FUNCTION_BLOCK ConveyorLL
VAR
	enable AT %Q* : BOOL := TRUE;
	direction AT %Q* : BOOL; //FALSE = forward, TRUE = backward
	pulse AT %Q* : BOOL;
	reset AT %Q* : BOOL;
	
	sensorEntry AT %I* : BOOL;
	sensorExit AT %I* : BOOL;

	lifterEnable AT %Q* : BOOL := TRUE;
	lifterDirection AT %Q* : BOOL; //FALSE = up, TRUE = down
	lifterPulse AT %Q* : BOOL;
	lifterReset AT %Q* : BOOL;
END_VAR
VAR_OUTPUT
	operation : ConveyorMode;
	request : ConveyorMode;
	
	error AT %I* : BOOL;
	lifterError AT %I* : BOOL;
	
	position AT %I* : REAL;
	velocity AT %I* : REAL;
	
	hasLifter : BOOL;
	extended AT %I* : BOOL;
	retracted AT %I* : BOOL;
END_VAR
VAR
	nextConveyor : POINTER TO Conveyor;
	prevConveyor : POINTER TO Conveyor;
	
	lifterMode : (HOLD, LIFTER_EXTEND, LIFTER_RETRACT); 
	
	//pulses are assumed to be low-high-low
	pulser : TP;
	lifterPulser : TP;
END_VAR
VAR_STAT CONSTANT
	pulseWidth : TIME := T#25MS;
END_VAR

pulser(IN:= , PT:= pulseWidth, Q=> pulse, ET=> );
pulser.IN := 
	enable AND 
	NOT error AND 
	NOT reset AND 
	(operation = ConveyorMode.FORWARD OR operation = ConveyorMode.BACKWARD)
	AND pulser.Q; //ends pulse itself

lifterPulser(IN:= , PT:= pulseWidth, Q=> lifterPulse, ET=> );
lifterPulser.IN := 
	hasLifter AND
	lifterEnable AND 
	NOT lifterError AND 
	NOT lifterReset AND 
	( (lifterMode = LIFTER_EXTEND AND NOT extended) OR (lifterMode = LIFTER_RETRACT AND NOT retracted) ) AND
	lifterPulser.Q; //self-ending pulse

override();

CASE lifterMode OF
	HOLD:
		lifterDirection := TRUE;
		lifterPulse := FALSE;
		
	LIFTER_EXTEND:
		lifterDirection := FALSE;
		lifterPulse := NOT lifterPulse;
	
	LIFTER_RETRACT:
		lifterDirection := TRUE;
		lifterPulse := NOT lifterPulse;
	
END_CASE

sequence();

METHOD backward : BOOL
VAR_INPUT
END_VAR
END_METHOD

METHOD extend : BOOL
VAR_INPUT
END_VAR
VAR
	noLifter : BOOL;
END_VAR
IF hasLifter THEN
	lifterMode := UP;
	extend := TRUE;
ELSE
	noLifter := TRUE;
END_IF
END_METHOD

METHOD forward : BOOL
VAR_INPUT
END_VAR
END_METHOD

PROPERTY IsOccupied : BOOL
GET
IsOccupied := sensorExit OR sensorEntry;
END_GET
END_PROPERTY

METHOD PRIVATE override : BOOL
VAR_INPUT
END_VAR
IF
	(extended AND lifterMode = UP) OR
	(retracted AND lifterMode = DOWN)
THEN
	lifterMode := HOLD;
END_IF
END_METHOD

METHOD reset : BOOL
VAR_INPUT
END_VAR
position := 0;
velocity := velocity; //no change

extend();
END_METHOD

METHOD retract : BOOL
VAR_INPUT
END_VAR
VAR
	noLifter : BOOL;
END_VAR
IF hasLifter THEN
	lifterMode := DOWN;
	retract := TRUE;
ELSE
	noLifter := TRUE;
END_IF
END_METHOD

METHOD PRIVATE sequence : BOOL
VAR_INPUT
END_VAR
VAR
	nextOp, prevOp : ConveyorMode;
END_VAR
IF nextConveyor <> 0 THEN
	nextOp := nextConveyor^.operation;
END_IF
IF prevConveyor <> 0 THEN
	prevOp := prevConveyor^.operation;
END_IF


IF IsOccupied THEN
	operation := MAX(nextOp, request, prevOp);
ELSE
	operation := ConveyorMode.IDLE;
END_IF


direction := (operation = ConveyorMode.BACKWARD); //set direction bit

IF hasLifter THEN
	
END_IF
END_METHOD

METHOD setOperation : BOOL
VAR_INPUT
	newOperation : ConveyorMode;
END_VAR
operation := newOperation;
END_METHOD

METHOD setRequest : BOOL
VAR_INPUT
	requestedMode : ConveyorMode;
END_VAR
request := requestedMode;
END_METHOD

METHOD target : BOOL
VAR_INPUT
	targetPosition : REAL;
END_VAR
END_METHOD

END_FUNCTION_BLOCK

(* stored: Version 1.1.0.1, ProductVersion 3.1.4024.11
   POU ConveyorLL: Id {fc7e9ede-e80d-4145-a9d9-be00ee3b7556}, SpecialFunc None
   Folder Properties: Id {d361e368-e054-4305-920b-b9dbf510eefd}
   Folder Unused: Id {be3cc95c-ce7d-4e3d-a436-a03da4486657}
   Method backward: Id {ca0e1347-ec46-44d4-8c44-e8bc9168c713}
   Method extend: Id {c91a1c6b-9055-436d-acf0-c83f5887a631}
   Method forward: Id {b7babf15-33c0-4022-a2f8-96a2d5ac67ee}
   Property IsOccupied: Id {861efb00-8fc8-4296-bd98-9ec5cf49340e}
   Get Get: Id {ba08d071-417b-4db9-b2e5-0b32fd8cd06d}
   Method override: Id {a607cbb0-0bbc-464a-85b1-298bf300cee2}
   Method reset: Id {1dd287fd-8076-405a-aa6b-b9bf311526be}
   Method retract: Id {4f15a35a-e7b6-4ba7-806b-8d9715fa3d20}
   Method sequence: Id {64079123-6890-47af-a137-de9efb652062}
   Method setOperation: Id {cd412fa0-1649-4a7d-925f-5d38574e0904}
   Method setRequest: Id {3d922abb-bb15-47df-a509-dc07d36b489c}
   Method target: Id {c8cd6c25-642c-4546-a8d0-1002f2e9247e} *)
